Fanuc KAREL source: kt00543.KL

-- PROVISIONAL review KL for V940-1; original PC SHA256 5479991b1244f650a173fe33f5e4b15bea373c3252efd979dccb09162ed3449e
-- Incomplete behavior may be omitted. Consult companion uncertainty JSON. Do not deploy.
PROGRAM KT00543
%NOLOCKGROUP
VAR
  OUT : BOOLEAN
-- UNRESOLVED_DECL P1 type=000199
-- UNRESOLVED_DECL P2 type=000106
BEGIN
  -- V9_ZERO_TABLE_METADATA_HINT layout=0001; no indexed target words; source/name/runtime held
  -- UNRESOLVED_PC offsets 5-20; opcodes 2E,22,32,35
  -- UNRESOLVED_PC offsets 25-58; opcodes 49,7E,49,7E,AC,23
  -- UNRESOLVED_PC offsets 63-67; opcodes 7F
END KT00543
